// Mitsubishi GX Works2 project: auto on; Auto rst   PLC: FX1N/FX1NC

PROGRAM MAIN
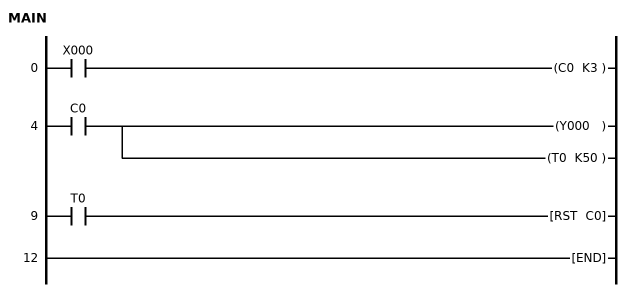
0     LD      X000
      OUT     C0 K3
4     LD      C0
      OUT     Y000
      OUT     T0 K50
9     LD      T0
      RST     C0
12    END
END_PROGRAM
